(* IEC 61131-3 sources: esstee/src/tests/programs/function_blocks, 15 files *)

(* ---- circular_ref.ST ---- *)
FUNCTION_BLOCK fb_s

VAR
	myself : fb_s;
END_VAR

;

END_FUNCTION_BLOCK

PROGRAM t

;

END_PROGRAM

(* ---- circular_ref_2.ST ---- *)
FUNCTION_BLOCK fb_1_s

VAR
	other_fb : fb_2_s;
END_VAR

;

END_FUNCTION_BLOCK

FUNCTION_BLOCK fb_2_s

VAR
	the_other_fb : fb_1_s;
END_VAR

;

END_FUNCTION_BLOCK

PROGRAM t

;

END_PROGRAM

(* ---- circular_ref_3.ST ---- *)
FUNCTION_BLOCK fb_1

VAR
	var_fb_1 : fb_2;
END_VAR

;

END_FUNCTION_BLOCK

FUNCTION_BLOCK fb_2

VAR
	var_fb_2 : fb_3;
END_VAR

;

END_FUNCTION_BLOCK

FUNCTION_BLOCK fb_3

VAR
	var_fb_3 : fb_1;
END_VAR

;

END_FUNCTION_BLOCK

PROGRAM t

;

END_PROGRAM

(* ---- circular_ref_4.ST ---- *)
TYPE
	d1 : fb_1;
	d2 : fb_2;
	d3 : fb_3;
END_TYPE

FUNCTION_BLOCK fb_1

VAR
	var_fb_1 : d1;
END_VAR

;

END_FUNCTION_BLOCK

FUNCTION_BLOCK fb_2

VAR
	var_fb_2 : d2;
END_VAR

;

END_FUNCTION_BLOCK

FUNCTION_BLOCK fb_3

VAR
	var_fb_3 : d3;
END_VAR

;

END_FUNCTION_BLOCK

PROGRAM t

;

END_PROGRAM

(* ---- circular_ref_5.ST ---- *)
TYPE
	d1 : fb_1;
	d2 : d3;
	d3 : d1;
END_TYPE

FUNCTION_BLOCK fb_1

VAR
	var_fb_1 : d1;
END_VAR

;

END_FUNCTION_BLOCK

FUNCTION_BLOCK fb_2

VAR
	var_fb_2 : d2;
END_VAR

;

END_FUNCTION_BLOCK

FUNCTION_BLOCK fb_3

VAR
	var_fb_3 : d3;
END_VAR

;

END_FUNCTION_BLOCK

PROGRAM t

;

END_PROGRAM

(* ---- circular_ref_6.ST ---- *)
TYPE
	d1 : fb_2;
	d2 : d3;
	d3 : d1;
END_TYPE

FUNCTION_BLOCK fb_1

VAR
	var_fb_1 : d1;
END_VAR

;

END_FUNCTION_BLOCK

FUNCTION_BLOCK fb_2

VAR
	var_fb_2 : d2;
END_VAR

;

END_FUNCTION_BLOCK

FUNCTION_BLOCK fb_3

VAR
	var_fb_3 : d3;
END_VAR

;

END_FUNCTION_BLOCK

PROGRAM t

;

END_PROGRAM

(* ---- conditionals.ST ---- *)
FUNCTION_BLOCK fb_if

VAR
	i1 : DINT;
	i2 : DINT;
END_VAR

if i1 = 1 then
   i2 := 10;
elsif i1 = 2 then
   i2 := 20;
elsif i1 = 3 then
   i2 := 30;
else
   i2 := 40;
end_if;

END_FUNCTION_BLOCK

PROGRAM t_if

VAR
	fb : fb_if;
END_VAR

fb();

END_PROGRAM

FUNCTION_BLOCK fb_case

VAR
	i1 : DINT;
	i2 : DINT;
END_VAR

case i1 of

1: i2 := 10;

2: i2 := 20;

3: i2 := 30;

else i2 := 40;

end_case;

END_FUNCTION_BLOCK

PROGRAM t_case

VAR
	fb : fb_case;
END_VAR

fb();

END_PROGRAM

(* ---- invoke.ST ---- *)
FUNCTION return_value : INT

VAR_INPUT
	val1 : INT;
	val2 : INT;
END_VAR

return_value := val1 + val2;

END_FUNCTION

FUNCTION_BLOCK test_fb

VAR_INPUT
	a : INT;
	b : INT;
END_VAR

VAR
	c : INT;
END_VAR

c := return_value(a, b);

END_FUNCTION_BLOCK

PROGRAM t

VAR
	fb : test_fb;
END_VAR

fb(1, 2);

END_PROGRAM

(* ---- loops.ST ---- *)
FUNCTION_BLOCK fb_for

VAR
	itr : INT;
	out : ARRAY[1..5] of INT;
	out2 : ARRAY[1..5] of INT;
END_VAR

for itr := 1 to 5 do
    out[itr] := itr;
    out2[itr] := itr * 2;
end_for;

END_FUNCTION_BLOCK

PROGRAM t_for

VAR
	fb : fb_for;
END_VAR

fb();

END_PROGRAM

FUNCTION_BLOCK fb_while

VAR
	itr : INT := 0;
	control : INT := 0;
	control_two : INT := 0;
	itr_two : INT := 0;
END_VAR

while True do
      itr := itr + 1;

      if itr > 5 then
      	 exit;
      end_if;

      control := control + 1;

end_while;

while False do
      control_two := 100;
end_while;

while itr_two < 4 do
      itr_two := itr_two + 1;
end_while;

END_FUNCTION_BLOCK

PROGRAM t_while

VAR
	fb : fb_while;
END_VAR

fb();

END_PROGRAM

FUNCTION_BLOCK fb_repeat

VAR
	itr : INT := 0;
	control : INT := 0;
	control_two : INT := 0;
	itr_two : INT := 0;
END_VAR

repeat
      itr := itr + 1;

      if itr > 5 then
      	 exit;
      end_if;

      control := control + 1;
until False
end_repeat;

repeat
      control_two := control_two + 1;
until True
end_repeat;

repeat
	itr_two := itr_two + 1;
until itr_two > 4
end_repeat;

END_FUNCTION_BLOCK

PROGRAM t_repeat

VAR
	fb : fb_repeat;
END_VAR

fb();

END_PROGRAM

(* ---- noninput.ST ---- *)
FUNCTION_BLOCK simple_s

VAR_INPUT
	in : INT;
END_VAR

;

END_FUNCTION_BLOCK

(* Assigning non-input variables *)
PROGRAM bad_non_input

VAR
	simple : simple_s;
END_VAR

simple(last:=1);

END_PROGRAM

(* ---- qualified_assignment.ST ---- *)
FUNCTION_BLOCK test_fb

VAR_INPUT
	ai : INT;
	bi : INT;
END_VAR

VAR
	a : ARRAY[1..5] of INT;
	b : ARRAY[1..5] of INT;
END_VAR

a[ai] := ai*100;
b[bi] := bi*100;

END_FUNCTION_BLOCK

PROGRAM t

VAR
	t1 : test_fb;
	t2 : test_fb;
END_VAR

t1(ai:=1, bi:=2);
t2(ai:=5, bi:=3);

END_PROGRAM

FUNCTION_BLOCK test_fb_nest

VAR
	t1 : test_fb;
END_VAR

t1(ai:=1, bi:=2);

END_FUNCTION_BLOCK

PROGRAM tnest

VAR
	t : test_fb_nest;
END_VAR

t();

END_PROGRAM

(* ---- simple.ST ---- *)
FUNCTION_BLOCK simple_s

VAR_INPUT
	in : INT;
END_VAR

VAR_OUTPUT
	out : INT;
END_VAR

VAR
	last : INT;
END_VAR

;

last := out;
out := last + in;

END_FUNCTION_BLOCK

(* Calling variable amount of times *)
PROGRAM t

VAR
	a : INT;
	b : INT;
	itr : INT;
	simple : simple_s;
END_VAR

for itr := 1 to b do
    simple(in:=a);
end_for;

END_PROGRAM

(* Calling without arguments *)
PROGRAM no_args

VAR
	simple : simple_s;
END_VAR

simple();

END_PROGRAM

(* Wrong type for in *)
PROGRAM bad_in_type

VAR
	simple : simple_s;
END_VAR

simple(in:=true and false);

END_PROGRAM

(* ---- simple_assignment.ST ---- *)
FUNCTION_BLOCK assign_s

VAR_INPUT
	in : INT;
END_VAR

VAR
	out : INT;
END_VAR

out := in;

END_FUNCTION_BLOCK

PROGRAM t

VAR
	a0 : assign_s;
	a1 : assign_s;
	a2 : assign_s;
	a3 : assign_s;
END_VAR

a1(10);
a2(20);

END_PROGRAM

PROGRAM t2

VAR
	a1 : assign_s;
END_VAR

;

END_PROGRAM

(* ---- toomany.ST ---- *)
FUNCTION_BLOCK simple_s

VAR_INPUT
	in1 : INT;
END_VAR

;

END_FUNCTION_BLOCK

(* Too many inputs *)
PROGRAM bad_too_many

VAR
	simple : simple_s;
END_VAR

simple(in1:=1, 10);

END_PROGRAM

(* ---- undefined.ST ---- *)
FUNCTION_BLOCK simple

;

END_FUNCTION_BLOCK

(* Undefined fb handle *)
PROGRAM bad_undefined

simple(in:=1);

END_PROGRAM
